// TwinCAT 3 PLC project Untitled1
// ProgramVersion: 3.1.4022.6
// libraries:
//   Tc2_MC2, * (Beckhoff Automation GmbH)
//   Tc2_Standard, * (Beckhoff Automation GmbH)
//   Tc2_System, * (Beckhoff Automation GmbH)
//   Tc3_Module, * (Beckhoff Automation GmbH)
// project tree:
//   DUTs/Servo/ AxisFn.TcDUT, MotionFn.TcDUT, StatParamFn.TcDUT, typ_ServoIF.TcDUT
//   DUTs/Servo/typMotion/ typ_MotionGearing.TcDUT, typ_MotionHoming.TcDUT, typ_MotionManualMotion.TcDUT, typ_MotionPhasing.TcDUT, typ_MotionPointToPoint.TcDUT
//   GVLs/ gc.TcGVL, gFB.TcGVL
//   / PlcTask.TcTTO
//   POUs/ MAIN.TcPOU
// real-time tasks:
//   TASK PlcTask: cycle T#10ms, priority 20, ADS port 350
// motion (NC):
//   TASK NC-Task 1 SAF: cycle T#2ms, priority 4, ADS port 501
//   TASK NC-Task 1 SVB: cycle T#10ms, priority 8, ADS port 511
//   AXIS Axis 1 (id 1)
//     General: UnitName=Degree
//     Dynamic: Acceleration=46989, Deceleration=46989, Jerk=140967
//     Velo: RefSearch=313.26, RefSync=313.26, SlowManual=1566.3, FastManual=9397.8, Fast=31326, Maximum=31326
//     OtherSettings: AllowMotionCmdToSlave=true
//     encoder EncType=19
//       EncPara: ScaleFactorNumerator=360, ScaleFactorDenominator=1048576, MaxCount=#xffffffff
//     drive DrvType=16
//       DrvPara: MaxCount=#xffffffff, DriveControlDWord=#x00020000
//         Analog: VeloReferenz=34458.6, VeloScale=32, ScaleFactorActTorque=0.1
//         TimeComp: TaskDelayCycles=1
//     controller CtrType=1
//       CtrPara: PriorControlFactor=1
//         Observer: BandWidth=20
//   AXIS Axis 2 (id 2)
//     General: UnitName=Degree
//     Dynamic: Acceleration=46989, Deceleration=46989, Jerk=140967
//     Velo: RefSearch=313.26, RefSync=313.26, SlowManual=1566.3, FastManual=9397.8, Fast=31326, Maximum=31326
//     OtherSettings: AllowMotionCmdToSlave=true
//     encoder EncType=19
//       EncPara: ScaleFactorNumerator=360, ScaleFactorDenominator=1048576, MaxCount=#xffffffff
//     drive DrvType=16
//       DrvPara: MaxCount=#xffffffff, DriveControlDWord=#x00020000
//         Analog: VeloReferenz=34458.6, VeloScale=32, ScaleFactorActTorque=0.1
//         TimeComp: TaskDelayCycles=1
//     controller CtrType=1
//       CtrPara: PriorControlFactor=1
//         Observer: BandWidth=20
// I/O:
//   DEVICE Device 1 (EtherCAT), AmsNetId 192.168.1.76.2.1
//     Term 1 (EK1828) [EK1828 EtherCAT IO-Coupler  (1A E-Bus, 4 Ch. Dig. In, 3ms, 8 Ch. Dig. Out 24V, 0,5A)]
//       Term 2 (EL3314) [EL3314 4Ch. Ana. Input Thermocouple (TC)]
//       Term 3 (EL3164) [EL3164 4Ch. Ana. Input 0-10V]
//       Term 4 (EL7201-9014) [EL7201-9014 1Ch. MDP742 Servo motor output stage with OCT (50V, 2.8A RMS) and STO input]
//       Term 5 (EL7201-9014) [EL7201-9014 1Ch. MDP742 Servo motor output stage with OCT (50V, 2.8A RMS) and STO input]
//       Term 6 (EL9011) [EL9011 End Terminal]
// variable links:
//   NC-Task 1 SAF/Axes/Axis 1 <-> Device 1 (EtherCAT)/Term 1 (EK1828)/Term 4 (EL7201-9014)
//     Drive/Inputs/In/nDcOutputTime <-> InfoData/DcOutputShift
//     Drive/Inputs/In/nState1 <-> DRV Statusword/Statusword
//     Drive/Inputs/In/nState2 <-> DRV Statusword/Statusword @bit 8
//     Drive/Inputs/In/nState4 @bit 1 <-> WcState/InputToggle
//     Drive/Inputs/In/nState4 <-> WcState/WcState
//     Drive/Outputs/Out/nCtrl1 <-> DRV Controlword/Controlword
//     Drive/Outputs/Out/nCtrl2 <-> DRV Controlword/Controlword @bit 8
//     Drive/Outputs/Out/nDataOut2 <-> DRV Target velocity/Target velocity
//     Enc/Inputs/In/nDataIn1 <-> FB Position/Position
//     Enc/Inputs/In/nDcInputTime <-> InfoData/DcInputShift
//     Enc/Inputs/In/nState4 @bit 1 <-> WcState/InputToggle
//     Enc/Inputs/In/nState4 <-> WcState/WcState
//   NC-Task 1 SAF/Axes/Axis 2 <-> Device 1 (EtherCAT)/Term 1 (EK1828)/Term 5 (EL7201-9014)
//     Drive/Inputs/In/nDcOutputTime <-> InfoData/DcOutputShift
//     Drive/Inputs/In/nState1 <-> DRV Statusword/Statusword
//     Drive/Inputs/In/nState2 <-> DRV Statusword/Statusword @bit 8
//     Drive/Inputs/In/nState4 @bit 1 <-> WcState/InputToggle
//     Drive/Inputs/In/nState4 <-> WcState/WcState
//     Drive/Outputs/Out/nCtrl1 <-> DRV Controlword/Controlword
//     Drive/Outputs/Out/nCtrl2 <-> DRV Controlword/Controlword @bit 8
//     Drive/Outputs/Out/nDataOut2 <-> DRV Target velocity/Target velocity
//     Enc/Inputs/In/nDataIn1 <-> FB Position/Position
//     Enc/Inputs/In/nDcInputTime <-> InfoData/DcInputShift
//     Enc/Inputs/In/nState4 @bit 1 <-> WcState/InputToggle
//     Enc/Inputs/In/nState4 <-> WcState/WcState
//   Untitled1/Untitled1 Instance <-> Device 1 (EtherCAT)/Term 1 (EK1828)
//     PlcTask Outputs/MAIN.xLamp <-> Channel 5/Output

CONFIGURATION Untitled1
    RESOURCE PLC ON TwinCAT3
        TASK PlcTask(INTERVAL := T#10ms, PRIORITY := 20);
        PROGRAM MAIN WITH PlcTask : MAIN;
    END_RESOURCE
END_CONFIGURATION

// ---- DUTs/Servo/AxisFn.TcDUT
TYPE AxisFn :
STRUCT
	MC_Power		: MC_Power;
	MC_Reset		: MC_Reset;
	MC_SetPosition	: MC_SetPosition;
END_STRUCT
END_TYPE

// ---- DUTs/Servo/MotionFn.TcDUT
TYPE MotionFn :
STRUCT
	Gearing						: typ_MotionGearing;
	Homing						: typ_MotionHoming;
	ManualMotion				: typ_MotionManualMotion;
	Phasing						: typ_MotionPhasing;
	PointToPoint				: typ_MotionPointToPoint;
END_STRUCT
END_TYPE

// ---- DUTs/Servo/typMotion/typ_MotionGearing.TcDUT
TYPE typ_MotionGearing :
STRUCT
	MC_GearIn					: MC_GearIn;
	MC_GearInDyn				: MC_GearInDyn;
	MC_GearInMultiMaster		: MC_GearInMultiMaster;
	MC_GearOut					: MC_GearOut;
END_STRUCT
END_TYPE

// ---- DUTs/Servo/typMotion/typ_MotionHoming.TcDUT
TYPE typ_MotionHoming :
STRUCT
	MC_Home						: MC_Home;
END_STRUCT
END_TYPE

// ---- DUTs/Servo/typMotion/typ_MotionManualMotion.TcDUT
TYPE typ_MotionManualMotion :
STRUCT
	MC_Jog				: MC_Jog;
END_STRUCT
END_TYPE

// ---- DUTs/Servo/typMotion/typ_MotionPhasing.TcDUT
TYPE typ_MotionPhasing :
STRUCT
	MC_HaltPhasing				: MC_HaltPhasing;
	MC_PhasingAbsolute			: MC_PhasingAbsolute;
	MC_PhasingRelative			: MC_PhasingRelative;
END_STRUCT
END_TYPE

// ---- DUTs/Servo/typMotion/typ_MotionPointToPoint.TcDUT
TYPE typ_MotionPointToPoint :
STRUCT
	MC_Halt						: MC_Halt;
	MC_MoveAbsolute				: MC_MoveAbsolute;
	MC_MoveAdditive				: MC_MoveAdditive;
	MC_MoveContinuousAbsolute	: MC_MoveContinuousAbsolute;
	MC_MoveContinuousRelative	: MC_MoveContinuousRelative;
	MC_MoveModulo				: MC_MoveModulo;
	MC_MoveRelative				: MC_MoveRelative;
	MC_MoveVelocity				: MC_MoveVelocity;
	MC_Stop						: MC_Stop;
END_STRUCT
END_TYPE

// ---- DUTs/Servo/StatParamFn.TcDUT
TYPE StatParamFn :
STRUCT
	MC_ReadActualPosition				: MC_ReadActualPosition;
	MC_ReadActualVelocity				: MC_ReadActualVelocity;
	MC_ReadAxisComponents				: MC_ReadAxisComponents;
	MC_ReadAxisError					: MC_ReadAxisError;
	MC_ReadBoolParameter				: MC_ReadBoolParameter;
	MC_ReadParameter					: MC_ReadParameter;
	MC_ReadParameterSet					: MC_ReadParameterSet;
	MC_ReadStatus						: MC_ReadStatus;
	MC_WriteBoolParameter				: MC_WriteBoolParameter;
	MC_WriteBoolParameterPersistent		: MC_WriteBoolParameterPersistent;
	MC_WriteParameter					: MC_WriteParameter;
	MC_WriteParameterPersistent			: MC_WriteParameterPersistent;
END_STRUCT
END_TYPE

// ---- DUTs/Servo/typ_ServoIF.TcDUT
TYPE typ_ServoIF :
STRUCT
	Axis_Ref								: AXIS_REF;
	Axis									: AxisFn;
	Motion									: MotionFn;
	StatParam								: StatParamFn;
END_STRUCT
END_TYPE

// ---- GVLs/gc.TcGVL
{attribute 'qualified_only'}
VAR_GLOBAL CONSTANT
	usiMaxNrOfAxes	: USINT	:= 2;
	usiAxisIndex1	: USINT	:= 0;
	usiAxisIndex2	: USINT	:= 1;
END_VAR

// ---- GVLs/gFB.TcGVL
{attribute 'qualified_only'}
VAR_GLOBAL
	arrServoCtrl			: ARRAY[0..gc.usiMaxNrOfAxes] OF typ_ServoIF;
END_VAR

// ---- POUs/MAIN.TcPOU
PROGRAM MAIN
VAR
	xSwitch			: BOOL;
	xLamp	AT %Q*	: BOOL;
	
	astServoIF		: ARRAY[0..gc.usiMaxNrOfAxes] OF typ_ServoIF;
END_VAR

xLamp	:= xSwitch;

END_PROGRAM
